(* IEC 61131-3 sources: Std_PalletMover/Class/_Settingsbase, 1 file *)

(* ---- _Settingsbase.st ---- *)
(*!
<Class
	Name               = "_Settingsbase"
	Revision           = "0.0"
	RealtimeTask       = "false"
	CyclicTask         = "false"
	BackgroundTask     = "false"
	Sigmatek           = "false"
	OSInterface        = "false"
	HighPriority       = "false"
	Automatic          = "false"
	UpdateMode         = "Prescan"
	SharedCommandTable = "true"
	Objectsize         = "(420,240)">
	<Channels>
		<Server Name="ClassSvr" Visualized="false" Initialize="false" WriteProtected="true" Retentive="false"/>
		<Server Name="ItemError" Visualized="false" Initialize="false" WriteProtected="true" Retentive="false"/>
		<Server Name="ItemOk" Visualized="false" Initialize="false" WriteProtected="true" Retentive="false"/>
		<Client Name="JsReader" Required="true" Internal="true"/>
		<Client Name="JsWriter" Required="true" Internal="true"/>
		<Client Name="op_LogData" Required="false" Internal="false" Comment="Output for logging data to SF_Logger"/>
		<Client Name="WewoBase3" Required="true" Internal="true"/>
	</Channels>
	<Network Name="_Settingsbase">
		<!-- List of Components in this network -->
		<Components>
			<Object
				Name           = "JsReader"
				Class          = "_JSONReader"
				Position       = "(780,210)"
				Visualized     = "true"
				Remotely       = "true"
				BackgroundTime = "10 ms">
				<Channels>
					<Server Name="ClassSvr"/>
					<Server Name="LibraryVersion"/>
					<Server Name="ReadFSM"/>
					<Client Name="_FileSys"/>
					<Client Name="SigCLib"/>
				</Channels>
			</Object>
			<Object
				Name           = "JsWriter"
				Class          = "_JSONWriter"
				Position       = "(180,210)"
				Visualized     = "true"
				Remotely       = "true"
				BackgroundTime = "10 ms">
				<Channels>
					<Server Name="ClassSvr"/>
					<Server Name="LibraryVersion"/>
					<Server Name="WriteFSM"/>
					<Client Name="_FileSys"/>
					<Client Name="SigCLib"/>
				</Channels>
			</Object>
			<Object
				Name       = "WewoBase3"
				Class      = "WewoBase"
				Position   = "(570,540)"
				Visualized = "false">
				<Channels>
					<Server Name="m_Id"/>
					<Server Name="m_p_Name"/>
					<Server Name="o_ErrorWarningStatus"/>
					<Server Name="ObjectStatus"/>
					<Server Name="ToObject"/>
					<Client Name="c_Group"/>
					<Client Name="op_LogData"/>
					<Client Name="toOsLibTaskObjControl"/>
				</Channels>
			</Object>
		</Components>
		<Comments>
		</Comments>
		<!-- List of Connections in this network -->
		<Connections>
			<Connection Source="this.JsReader" Destination="JsReader.ClassSvr"/>
			<Connection Source="this.JsWriter" Destination="JsWriter.ClassSvr"/>
			<Connection Source="this.WewoBase3" Destination="WewoBase3.ToObject"/>
			<Connection Source="WewoBase3.op_LogData" Destination="this.op_LogData" Vertices="(570,630),(38,210),"/>
		</Connections>
		<!-- Headerfiles -->
		<Options>
		</Options>
	</Network>
</Class>
*)
_Settingsbase : CLASS
  //Servers:
	ClassSvr 	: SvrChCmd_DINT;
	ItemOk 	: SvrCh_DINT;
	ItemError 	: SvrCh_DINT;
  //Clients:
	JsReader 	: CltChCmd__JSONReader;
	JsWriter 	: CltChCmd__JSONWriter;
	WewoBase3 	: CltChCmd_WewoBase;
	op_LogData 	: CltCh_gpt_LogData;
  //Variables:
		pObjectHandle 	: ^_cJSON::t_s_cJSON;
  //Functions:

	FUNCTION VIRTUAL GLOBAL Init;

	FUNCTION UpdateFile
		VAR_INPUT
			Name 	: ^CHAR;
		END_VAR
		VAR_OUTPUT
			Value 	: BOOL;
		END_VAR;

	FUNCTION Method;

	FUNCTION GLOBAL GetObjectPath
		VAR_INPUT
			Path 	: ^CHAR;
		END_VAR
		VAR_OUTPUT
			GetValue 	: ^_cJSON::t_s_cJSON;
		END_VAR;

	FUNCTION GLOBAL GetDintValue
		VAR_INPUT
			Path 	: ^CHAR;
		END_VAR
		VAR_OUTPUT
			value 	: DINT;
		END_VAR;

	FUNCTION GLOBAL GetStringValue
		VAR_INPUT
			Path 	: ^CHAR;
		END_VAR
		VAR_OUTPUT
			value 	: ^CHAR;
		END_VAR;

	FUNCTION GLOBAL GetDoubleValue
		VAR_INPUT
			Path 	: ^CHAR;
		END_VAR
		VAR_OUTPUT
			value 	: REAL;
		END_VAR;

	FUNCTION GLOBAL GetBooleanValue
		VAR_INPUT
			Path 	: ^CHAR;
		END_VAR
		VAR_OUTPUT
			value 	: BOOL;
		END_VAR;
  //Tables:
	FUNCTION @STD
		VAR_OUTPUT
			ret_code	: CONFSTATES;
		END_VAR;
	FUNCTION GLOBAL TAB @CT_;
END_CLASS;

#pragma using _JSONReader
#pragma using _JSONWriter
#pragma using WewoBase

FUNCTION _Settingsbase::UpdateFile
	VAR_INPUT
		Name 	: ^CHAR;
	END_VAR
	VAR_OUTPUT
		Value 	: BOOL;
	END_VAR

  Name:="c:\settings\Configuration.json";

    Value :=JsReader.ReadFile(Name) ;
    if Value = TRUE then
        pObjectHandle := JsReader.GetMainElement();
        ItemOk      :=  0;
        ItemError   :=  0;
        else

    end_if;

END_FUNCTION

FUNCTION _SettingsBase::Method

END_FUNCTION

FUNCTION GLOBAL _Settingsbase::GetObjectPath
	VAR_INPUT
		Path 	: ^CHAR;
	END_VAR
	VAR_OUTPUT
		GetValue 	: ^_cJSON::t_s_cJSON;
	END_VAR

    var
        LenString : dint;
        counter :dint;
        LocString : array[0..255] of CHAR;
        pos:byte;
        curchar :char;
    END_VAR

   LenString :=  _strlen(src:=Path)$dint;
   Counter := 0;
   GetValue :=  pObjectHandle;

    for  pos := 0 to LenString$dint do
        curchar :=  (path+pos)^ ;

        if (curchar = '.') | (curchar = 0)  | (curchar = '\') | (curchar = '/' ) then
            LocString[counter] := 0;
            if counter > 0 then
                GetValue := JsReader.GetObjectItem(object:=GetValue , string:=#LocString[0]);
                if pObjectHandle = nil then
                    exit;
                end_if;
            End_if;
            Counter :=0;
        else
            LocString[Counter] :=  curchar;
            Counter += 1;
        end_if;
    end_for;

    if GetValue <> nil then
       ItemOk += 1;
    else
       ItemError += 1;
    end_if;
END_FUNCTION

FUNCTION GLOBAL _Settingsbase::GetDintValue
	VAR_INPUT
		Path 	: ^CHAR;
	END_VAR
	VAR_OUTPUT
		value 	: DINT;
	END_VAR

    VAR
    	pReadVariableHandle  : ^_cJSON::t_s_cJSON;
    END_VAR

    pReadVariableHandle := GetObjectPath(Path);
    if pReadVariableHandle <> nil then
        value := pReadVariableHandle^.Val_Int$Dint;
    else
        WewoBase3.WriteActiveErrorWarning(IntErrorWarningId:=::gt_AgvErrors::SettingNotFound, LogLevel:=::gt_LogLevel::LL_ERROR_INTERNAL, p_msg:=Path);
    end_if;

END_FUNCTION

FUNCTION GLOBAL _Settingsbase::GetStringValue
	VAR_INPUT
		Path 	: ^CHAR;
	END_VAR
	VAR_OUTPUT
		value 	: ^CHAR;
	END_VAR

    VAR
    	pReadVariableHandle  : ^_cJSON::t_s_cJSON;
    END_VAR

    pReadVariableHandle := GetObjectPath(Path);
    if pReadVariableHandle <> nil then
        value := pReadVariableHandle^.Val_String$^char;
        else
        value := nil;
        WewoBase3.WriteActiveErrorWarning(IntErrorWarningId:=::gt_AgvErrors::SettingNotFound, LogLevel:=::gt_LogLevel::LL_ERROR_INTERNAL, p_msg:=Path);
    end_if;

END_FUNCTION

FUNCTION GLOBAL _Settingsbase::GetDoubleValue
	VAR_INPUT
		Path 	: ^CHAR;
	END_VAR
	VAR_OUTPUT
		value 	: REAL;
	END_VAR

    VAR
    	pReadVariableHandle  : ^_cJSON::t_s_cJSON;
       temp:dint;
    END_VAR

    value := 0;

    pReadVariableHandle := GetObjectPath(Path);
    if pReadVariableHandle <> nil then
        temp :=pReadVariableHandle^.Val_String$dint;
          else
        WewoBase3.WriteActiveErrorWarning(IntErrorWarningId:=::gt_AgvErrors::SettingNotFound, LogLevel:=::gt_LogLevel::LL_ERROR_INTERNAL, p_msg:=Path);
    end_if;

    value := to_real(temp);
END_FUNCTION

FUNCTION VIRTUAL GLOBAL _Settingsbase::Init

END_FUNCTION

FUNCTION GLOBAL _Settingsbase::GetBooleanValue
	VAR_INPUT
		Path 	: ^CHAR;
	END_VAR
	VAR_OUTPUT
		value 	: BOOL;
	END_VAR
       VAR
    	pReadVariableHandle  : ^_cJSON::t_s_cJSON;
        temp : ^char;
    END_VAR

      value := false;

    pReadVariableHandle := GetObjectPath(Path);
    if pReadVariableHandle <> nil then
        if pReadVariableHandle^.Val_String <> nil then
        _strupr(str:=pReadVariableHandle^.Val_String);
           if _stricmp(pReadVariableHandle^.Val_String ,temp) = 0 then
            value := true;
            else
            Value := false;
          end_if;
      end_if;
      else
                WewoBase3.WriteActiveErrorWarning(IntErrorWarningId:=::gt_AgvErrors::SettingNotFound, LogLevel:=::gt_LogLevel::LL_ERROR_INTERNAL, p_msg:=Path);
            value := false;
            // write error
     end_if;

END_FUNCTION
